FUNCTION_BLOCK GenericStagingTable EXTENDS GenericMaterialHolder
VAR_OUTPUT
	//hmiSlots : ARRAY[1..numSlots] OF MaterialSlot;
END_VAR
VAR
	i : DINT(1..10);
END_VAR
VAR_STAT CONSTANT
	numSlots : UINT := SIZEOF(tableSlotsA21Left)/SIZEOF(tableSlotsA21Left[1]);
END_VAR

SUPER^();
(*
FOR i:=LOWER_BOUND(slots, 1) TO UPPER_BOUND(slots, 1) BY 1 DO
	hmiSlots[i].material := slots[i];
	hmiSlots[i].occupied := occupied[i];
END_FOR
*)

METHOD autofill : BOOL
VAR_INPUT
	materialID : STRING;
END_VAR
VAR
	i : INT;
	slot : INT;
END_VAR
(*
this method will automatically find an open slot
*)
IF isFull() OR materialID = '' THEN
	RETURN;
END_IF

IF findOpenSlot(materialID, openSlot=> slot) THEN
	place(slot, materialID);
	autofill := TRUE;
	
	//ADSLOGSTR(msgCtrlMask := ADSLOG_MSGTYPE_ERROR , msgFmtStr := 'autofill: %s', strArg := materialID);
END_IF
END_METHOD

METHOD findOpenSlot : BOOL
VAR_INPUT
	materialID : STRING;
END_VAR
VAR_OUTPUT
	openSlot : INT := 0;
END_VAR
VAR
	i : INT;
END_VAR
IF FIND(materialID, 'WDW') > 0 THEN //top wide, load in slot 9-10
	FOR i:=9 TO 10 BY 1 DO
		IF slots[i] = '' THEN
			findOpenSlot := TRUE;
			openSlot := i;
			RETURN;
		END_IF
	END_FOR
	
//ELSIF FIND(materialID, 'WDT') > 0 OR FIND(materialID, 'WDS') > 0 THEN //standard width, load in slot 3-10
ELSIF FIND(materialID, 'WD') > 0 THEN //standard width, load in slot 1-8
	FOR i:=1 TO 8 BY 1 DO
		IF slots[i] = '' THEN
			findOpenSlot := TRUE;
			openSlot := i;
			RETURN;
		END_IF
	END_FOR
	
END_IF
END_METHOD

METHOD findSlot : BOOL
VAR_INPUT
	materialID : STRING;
END_VAR
VAR_OUTPUT
	atSlot : INT;
END_VAR
VAR
	i : INT;
END_VAR
FOR i:=1 TO numSlots BY 1 DO
	IF slots[i] = materialID THEN
		atSlot := i;
		findSlot := TRUE;
		RETURN;
	END_IF
END_FOR
END_METHOD

METHOD isEmpty : BOOL
VAR
	i : INT;
	temp : BOOL;
END_VAR
FOR i:=1 TO numSlots BY 1 DO
	temp := temp OR occupied[i]; //TRUE if any slots are occupied
END_FOR

isEmpty := NOT temp; //invert result - FALSE if any slots are occupied
END_METHOD

METHOD isFull : BOOL
VAR
	i : INT;
	temp : BOOL := TRUE;
END_VAR
FOR i:=1 TO numSlots BY 1 DO
	temp := temp AND occupied[i];
END_FOR

isFull := temp;
END_METHOD

METHOD place : BOOL
VAR_INPUT
	i : INT;
	materialID : STRING;
END_VAR
IF slots[i] = '' THEN
	slots[i] := materialID;
	place := TRUE;
END_IF
END_METHOD

METHOD remove : BOOL
VAR_INPUT
	i : INT;
END_VAR
VAR_OUTPUT
	materialID : STRING;
END_VAR
remove := slots[i] <> '';

materialID := slots[i];
slots[i] := '';
END_METHOD

END_FUNCTION_BLOCK

(* stored: Version 1.1.0.1, ProductVersion 3.1.4024.11
   POU GenericStagingTable: Id {86f30268-c033-4b26-ab89-12e7cd4acf96}, SpecialFunc None
   Method autofill: Id {85f89965-dfb3-421e-9fdd-f8a8434c5c09}
   Method findOpenSlot: Id {70b64d97-b0dd-4604-bcf4-e5f1f840892d}
   Method findSlot: Id {6eb1e5d2-5dfb-4973-9008-93aea3b02a25}
   Method isEmpty: Id {853383cf-82c8-43ea-b031-c9c33787565e}
   Method isFull: Id {debc6f61-e9f5-4fcf-9975-806ae5e84cf7}
   Method place: Id {bb7401bd-65d3-4fcc-bcf4-393f54f9df10}
   Method remove: Id {3a843bdc-d585-4891-a014-f6828230b4c8} *)
